{attribute addProperty BoxType "EJ2128-0000-0016"}
{attribute addProperty Id "ChannelAT %Q*ARRAY[0..7] OF Channel_7F374EB06480WcStateAT %I*WcState_28A8677510.1250InfoDataAT %I*InfoData_192954DE1620"}
{attribute addProperty CRC "1482585628"}
{attribute addProperty SizeInBites "81"}
{attribute addProperty SizeInBytes "10.125"}
TYPE EJ2128_A854BE6D :
STRUCT
	{attribute addProperty Name "Channel"}
	Channel : ARRAY[0..7] OF Channel_7F374EB0;
	{attribute addProperty Name "WcState"}
	WcState : WcState_28A86775;
	{attribute addProperty Name "InfoData"}
	InfoData : InfoData_192954DE;
END_STRUCT
END_TYPE

(* stored: Version 1.2.0.0, ProductVersion 3.1.4024.9
   DUT EJ2128_A854BE6D: Id {85ee3ae1-97a4-4f53-890c-ae20c32767cd} *)
